(*************************************** EtherCAT Diag *********************************************)
(* generate Net Id *)
sEcMasterNetId := F_CreateAmsNetId(nIds := arrEcMasterNetId);
fbEtherCATDiag(
    sIPCNetID			:= '',
    sMasterNetID		:= sEcMasterNetId,
    nMasterDevID		:= nEcMasterDeviceId,
    nSlaveCount			:= nEcMasterSlaveCount,
    nSlaveCountCfg		:= nEcMasterSlaveCountCfg,
    nMasterDevState		:= nEcMasterDevState,
    bAllFrameWcStatesOK	:= bAllFrameWcStatesOK,
    tTimeout			:= T#5s,
    astDiagSlaveInfo	:= astDiagSlaveInfo,
    astDiagSlaveInfoScanned	:= astDiagSlaveInfoScanned,
    bEtherCATOK			=> bEtherCATOK,
    bFrameWcStateError	=> bFrameWcStateError,
    bSlaveCountError	=> bSlaveCountError,
    bMasterDevStateError=> bMasterDevStateError,
    stMasterDevState	=> stMasterDevState,
    bBusy				=> bBusy,
    bError				=> bError,
    nErrorID			=> nErrorID
);

END_FUNCTION_BLOCK

// ---- POUs/Diagnostics/FB_EtherCATFrameDiag.TcPOU
FUNCTION_BLOCK FB_EtherCATFrameDiag
VAR_INPUT
    nFrmXWcState 		: WORD;				// FrmXWcState
    nReqZeroMask 		: WORD := 16#FFFF;	// mask, bit TRUE: require wFrmXWcState.bit = FALSE, bit FALSE: ignore wFrmXWcState.bit *)
END_VAR
VAR_OUTPUT
    bFrameWcStateOK		: BOOL;				// result of fram state check
END_VAR
VAR
END_VAR

(* mask out ignored error bits and compare result against 0 *)
bFrameWcStateOK := ((nFrmXWcState AND nReqZeroMask) = 0);

END_FUNCTION_BLOCK

// ---- POUs/Diagnostics/FB_EtherCATDiag.TcPOU
FUNCTION_BLOCK FB_EtherCATDiag
VAR_INPUT
    sIPCNetID					: T_AmsNetId; 	// AmsNetId of the IPC
    sMasterNetID				: T_AmsNetId; 	// AmsNetId of the EtherCAT master device
    nMasterDevID				: UINT;			// Device ID of EtherCAT master
    nSlaveCount 				: UINT;			// current slave count
    nSlaveCountCfg 				: UINT;			// configured slave count
    nMasterDevState				: WORD;			// device state of EtherCAT Master
    bAllFrameWcStatesOK			: BOOL;			// all FrameWcState OK?
    tTimeout					: TIME := T#5S; // ads timeout
    eSubSystem : E_Subsystem := E_Subsystem.FIELDBUS; // Subsystem, change to (MPS, VACUUM, MOTION, etc)
END_VAR
VAR_OUTPUT
    bEtherCATOK					: BOOL;			// no problem on EtherCAT
    bFrameWcStateError			: BOOL;			// error in at least one frame
    bSlaveCountError			: BOOL;			// EtherCAT slave count mismatch (# of cfg slaves <> # of found slaves)
    bMasterDevStateError		: BOOL;			// error in master device state
    stMasterDevState			: ST_EcMasterDevState; // splitted master device state
    bBusy						: BOOL;			// FB busy
    bError						: BOOL;			// FB with error
    nErrorID					: UDINT;		// FB error ID
END_VAR
VAR_IN_OUT
    astDiagSlaveInfo 			: ARRAY [0..cnEscMaxPorts] OF ST_SlaveStateInfo;		// read in info from configured slaves
    astDiagSlaveInfoScanned		: ARRAY [0..cnEscMaxPorts] OF ST_SlaveStateInfoScanned;	// read in info from scanned slaves
END_VAR
VAR
    eState						: E_EcatDiagState;
    nMasterDevStatePrev			: WORD;
    bSlaveCountErrorPrev		: BOOL;
    bAllFrameWcStatesOKPrev		: BOOL;
    bDiagReq					: BOOL := TRUE;
    nI							: UDINT;
    nP							: UDINT;

    astSlaveInfo 				: ARRAY [0..cnSlaveAddrArrSize] OF ST_SlaveStateInfo;
    stSlaveInfo  :   REFERENCE TO ST_SlaveStateInfo;

    (* -- Get Slave Addresses *)
    fbGetSlaveAddresses 		: FB_EcGetAllSlaveAddr;
    anSlaveAddresses 			: ARRAY[0..cnSlaveAddrArrSize] OF UINT;
    nNumOfSlavesRead			: UINT;

    (* -- Get Slave States *)
    fbGetAllSlaveStates			: FB_EcGetAllSlaveStates;
    astSlaveStates 				: ARRAY[0..cnSlaveAddrArrSize] OF ST_EcSlaveState;

    (* -- Get Topology Data *)
    nTopologyData				: UDINT;
    fbGetTopologyData			: ADSREAD;
    astTopologyData				: ARRAY[0..cnSlaveAddrArrSize] OF ST_TopologyData;

    (* -- Check Topology *)
    anDiagIndex					: ARRAY [0..cnEscMaxPorts] OF UINT;
    nDiagIndex : UINT;
    anDiagPort					: ARRAY [0..cnEscMaxPorts] OF UINT;
    nDiagPort : UINT;
    nIdx						: DINT;

    (* -- Scan Slaves *)
    fbEcGetScannedSlaves		: FB_EcGetScannedSlaves;
    astScannedSlaveInfo			: ARRAY [0..cnSlaveAddrArrSize] OF ST_EcSlaveScannedData; // what...
    rScannedSlaveInfo   :   REFERENCE TO ST_EcSlaveScannedData;
    nScannedSlaves				: UINT;

    (* -- Get Slave Identities *)
    fbGetSlaveIdentity			: FB_EcGetSlaveIdentity;
    stIdentity 					: ST_EcSlaveIdentity;

    (* -- Get Slave Names *)
    fbGetSlaveName 				: IOF_GetBoxNameByAddr;
    astSlaveInfoScanned			: ARRAY [0..cnSlaveAddrArrSize] OF ST_SlaveStateInfoScanned; // the F
    stSlaveInfoScanned   :   REFERENCE TO ST_SlaveStateInfoScanned;
    sStringName						: STRING;



    // Logging components
    fbLogger : FB_LogMessage := (eSubsystem := eSubsystem);

    fbJson : FB_JsonSaxWriter;
    fbJsonDataType : FB_JsonReadWriteDataType;
    stDiagSlaveInfo : REFERENCE TO ST_SlaveStateInfo;
    fbEtherCATOK : F_TRIG;
    fbFrameWcStateError : R_TRIG;
    fbMasterError : R_TRIG;
    nJsonIdx : UINT;
    {attribute 'analysis' := '-27'}
    sTest : T_MaxString;
END_VAR

(* cyclic diag *)
bFrameWcStateError := NOT bAllFrameWcStatesOK;

bSlaveCountError := (nSlaveCount <> nSlaveCountCfg) OR (nSlaveCount = 0);
IF (bSlaveCountError AND NOT bSlaveCountErrorPrev) OR (NOT bSlaveCountError AND bSlaveCountErrorPrev) THEN
    bSlaveCountErrorPrev := bSlaveCountError;
    bDiagReq := TRUE; // slave count error change detected --> diag required
END_IF

IF (bAllFrameWcStatesOK AND NOT bAllFrameWcStatesOKPrev) OR (NOT bAllFrameWcStatesOK AND bAllFrameWcStatesOKPrev) THEN
    bAllFrameWcStatesOKPrev := bAllFrameWcStatesOK;
    bDiagReq := TRUE; // frame error change detected --> diag required
END_IF

IF (nMasterDevState <> nMasterDevStatePrev) THEN
    M_CheckMasterDevState();
    bDiagReq := TRUE; // devstate change detected --> diag required
END_IF

(* acyclic diag *)
CASE eState OF
E_EcatDiagState.Idle: (* IDLE *)
    IF bDiagReq THEN				// diag requested
        bDiagReq := FALSE;

        IF sMasterNetID <> '' AND sMasterNetID <> '0.0.0.0.0.0' THEN
            eState := E_EcatDiagState.GetSlaveAddresses;	// execute diag
            bBusy := TRUE;
        ELSE
            bError := TRUE;
            nErrorID := 7;
        END_IF

        bEtherCATOK := FALSE;
    ELSE
        // check for changes in idle
        IF (bSlaveCountError OR bMasterDevStateError OR NOT bAllFrameWcStatesOK) AND NOT (astSlaveInfo[anDiagIndex[0]].bDiagData) THEN
            bEtherCATOK := FALSE;
            bDiagReq := TRUE;//new error --> diag requested
        ELSIF (bSlaveCountError AND NOT bSlaveCountErrorPrev) OR (NOT bSlaveCountError AND bSlaveCountErrorPrev) THEN
            bSlaveCountErrorPrev := bSlaveCountError;
            bEtherCATOK := FALSE;
            bDiagReq := TRUE;// slave count error change detected --> diag required
        ELSIF (nMasterDevState <> nMasterDevStatePrev) THEN
            bEtherCATOK := FALSE;
            bDiagReq := TRUE;// devstate change detected --> diag required
        ELSIF (bAllFrameWcStatesOK AND NOT bAllFrameWcStatesOKPrev) OR (NOT bAllFrameWcStatesOK AND bAllFrameWcStatesOKPrev) THEN
            bAllFrameWcStatesOKPrev := bAllFrameWcStatesOK;
            bEtherCATOK := FALSE;
            bDiagReq := TRUE;// frame error change detected --> diag required
        ELSIF (bSlaveCountError OR bMasterDevStateError OR NOT bAllFrameWcStatesOK OR astSlaveInfo[anDiagIndex[0]].bDiagData) THEN
            bEtherCATOK := FALSE;
        ELSE
            bEtherCATOK := TRUE;
        END_IF
    END_IF

E_EcatDiagState.GetSlaveAddresses: (* get adresses *)
    M_GetSlaveAdresses();

E_EcatDiagState.GetSlaveStates: (* get states *)
    M_GetSlaveStates();

E_EcatDiagState.GetTopoDataLen:	(* get topology data length *)
    M_GetTopoDataLen();

E_EcatDiagState.GetTopoData:	(* get topology data *)
    M_GetTopoData();

E_EcatDiagState.ScanSlaves:	(* scan slaves *)
    M_ScanSlaves();

E_EcatDiagState.GetSlaveIdentity:	(* get identity *)
    M_GetSlaveIdentity();

E_EcatDiagState.GetSlaveName:	(* get name *)
    M_GetSlaveName();

E_EcatDiagState.GetScannedSlaveName:	(* get scanned name *)
    M_GetScannedSlaveName();

E_EcatDiagState.LogDiagnostics: (* Log diagnostics *)
    (* I can't get the fbJsonDataType to actually convert the slave info
    structures. I just get nulls. Either I am doing this wrong, or when
    the symbol parser encounters datatypes it can't deal with it nulls
    the whole thing. I'll keep this code commented out until someone figures
    out how to deal with parsing the slave structs into the json payload *)
    IF nJsonIdx < nNumOfSlavesRead THEN // the last entry is always blank
        nJsonIdx := MIN(cnSlaveAddrArrSize, nJsonIdx);
        stDiagSlaveInfo REF= astSlaveInfo[nJsonIdx];
        DiagnosticJson();
        fbLogger(sMsg:=CONCAT('Diag Results: ', stDiagSlaveInfo.sName),
                eSevr:=TcEventSeverity.Info);
        nJsonIdx := nJsonIdx + 1;
    ELSE
        nJsonIdx := 0;
        eState := E_EcatDiagState.Done;
    END_IF

E_EcatDiagState.Done:	(* DONE *)
    bBusy := FALSE;
    eState := 0;

END_CASE

// Log messages
fbEtherCATOK(CLK:=bEtherCATOK);
IF fbEtherCATOK.Q THEN
    fbLogger(sMsg:='EtherCAT failure, starting diagnostic', eSevr:=TcEventSeverity.Critical, sJson:='');
END_IF

fbFrameWcStateError(CLK:=bFrameWcStateError);
IF fbFrameWcStateError.Q THEN
    fbLogger(sMsg:='Working Counter Frame Error: error in at least one frame', eSevr:=TcEventSeverity.Error, sJson:='');
END_IF

fbMasterError(CLK:=bMasterDevStateError);
IF fbMasterError.Q THEN
    fbJson.StartObject();
        fbJson.AddKey('ecat_master_diag');
        fbJson.StartObject();
            fbJson.AddKey('bAtLeastOneNotInOp');
            fbJson.AddBool(stMasterDevState.bAtLeastOneNotInOp);
            fbJson.AddKey('bDcNotInSync');
            fbJson.AddBool(stMasterDevState.bDcNotInSync);
            fbJson.AddKey('bDriverNotFound');
            fbJson.AddBool(stMasterDevState.bDriverNotFound);
            fbJson.AddKey('bLinkError');
            fbJson.AddBool(stMasterDevState.bLinkError);
            fbJson.AddKey('bMissFrmRedMode');
            fbJson.AddBool(stMasterDevState.bMissFrmRedMode);
            fbJson.AddKey('bResetActive');
            fbJson.AddBool(stMasterDevState.bResetActive);
            fbJson.AddKey('bResetRequired');
            fbJson.AddBool(stMasterDevState.bResetRequired);
            fbJson.AddKey('bWatchdogTriggerd');
            fbJson.AddBool(stMasterDevState.bWatchdogTriggerd);
            fbJson.AddKey('eEcState');
            fbJson.AddUdint(stMasterDevState.eEcState);
        fbJson.EndObject();
    fbJson.EndObject();
    fbJson.CopyDocument(fbLogger.sJson, SIZEOF(fbLogger.sJson));
    fbLogger(sMsg:='Master error: error in master device state', eSevr:=TcEventSeverity.Critical);
    fbJson.ResetDocument();
END_IF

ACTION DiagnosticJson:
fbJson.StartObject();
    fbJson.AddKey('ecat_diag');
    fbJson.StartObject();

        fbJson.AddKey('nECAddr');
        fbJson.AddUdint(stDiagSlaveInfo.nECAddr);

        fbJson.AddKey('nIndex');
        fbJson.AddDint(stDiagSlaveInfo.nIndex);

        fbJson.AddKey('sName');
        fbJson.AddString(stDiagSlaveInfo.sName);

        fbJson.AddKey('sType');
        fbJson.AddString(stDiagSlaveInfo.sType);

        fbJson.AddKey('bDiagData');
        fbJson.AddBool(stDiagSlaveInfo.bDiagData);

        fbJson.AddKey('stPortCRCErrors');
        fbjson.StartObject();

            fbJson.AddKey('portA');
            fbJson.AddUdint(stDiagSlaveInfo.stPortCRCErrors.portA);
            fbJson.AddKey('portB');
            fbJson.AddUdint(stDiagSlaveInfo.stPortCRCErrors.portB);
            fbJson.AddKey('portC');
            fbJson.AddUdint(stDiagSlaveInfo.stPortCRCErrors.portC);
            fbJson.AddKey('portD');
            fbJson.AddUdint(stDiagSlaveInfo.stPortCRCErrors.portD);

        fbJson.EndObject();

        fbJson.AddKey('nSumCRCErrors');
        fbjson.AddUdint(stDiagSlaveInfo.nSumCRCErrors);

        fbJson.AddKey('stState');
        fbJson.StartObject();

            fbJson.AddKey('eEcState ');
            fbJson.AddUdint(stDiagSlaveInfo.stState.eEcState);
            fbJson.AddKey('nReserved');
            fbJson.AddUdint(stDiagSlaveInfo.stState.nReserved);
            fbJson.AddKey('bError');
            fbJson.AddBool(stDiagSlaveInfo.stState.bError);
            fbJson.AddKey('bInvalidVPRS');
            fbJson.AddBool(stDiagSlaveInfo.stState.bInvalidVPRS);
            fbJson.AddKey('nReserved2');
            fbJson.AddUdint(stDiagSlaveInfo.stState.nReserved2);
            fbJson.AddKey('bNoCommToSlave');
            fbJson.AddBool(stDiagSlaveInfo.stState.bNoCommToSlave);
            fbJson.AddKey('bLinkError');
            fbJson.AddBool(stDiagSlaveInfo.stState.bLinkError);
            fbJson.AddKey('bMissingLink');
            fbJson.AddBool(stDiagSlaveInfo.stState.bMissingLink);
            fbJson.AddKey('bUnexpectedLink');
            fbJson.AddBool(stDiagSlaveInfo.stState.bUnexpectedLink);
            fbJson.AddKey('bPortA');
            fbJson.AddBool(stDiagSlaveInfo.stState.bPortA);
            fbJson.AddKey('bPortB');
            fbJson.AddBool(stDiagSlaveInfo.stState.bPortB);
            fbJson.AddKey('bPortC');
            fbJson.AddBool(stDiagSlaveInfo.stState.bPortC);
            fbJson.AddKey('bPortD');
            fbJson.AddBool(stDiagSlaveInfo.stState.bPortD);

        fbJson.EndObject();

    fbJson.EndObject();

fbJson.EndObject();

fbJson.CopyDocument(fbLogger.sJson, SIZEOF(fbLogger.sJson));
fbJson.ResetDocument();
END_ACTION

ACTION M_CheckMasterDevState:
(* check master errors based on devstate *)
bMasterDevStateError 				:= nMasterDevState <> 0;
stMasterDevState.bLinkError 		:= ((nMasterDevState AND 16#000F) = 1) OR ((nMasterDevState AND 16#000F) = 4);
stMasterDevState.bResetRequired 	:= ((nMasterDevState AND 16#000F) = 2) OR ((nMasterDevState AND 16#FFF0) = 16#10);
stMasterDevState.bMissFrmRedMode 	:= (nMasterDevState AND 16#000F) = 8;
stMasterDevState.bWatchdogTriggerd 	:= (nMasterDevState AND 16#20) = 16#20;
stMasterDevState.bDriverNotFound 	:= (nMasterDevState AND 16#40) = 16#40;
stMasterDevState.bResetActive 		:= (nMasterDevState AND 16#80) = 16#80;
stMasterDevState.bAtLeastOneNotInOp := ((nMasterDevState AND 16#100) = 16#100) OR ((nMasterDevState AND 16#200) = 16#200) OR
                                        ((nMasterDevState AND 16#400) = 16#400) OR ((nMasterDevState AND 16#800) = 16#800);
stMasterDevState.bDcNotInSync 		:= (nMasterDevState AND 16#1000) = 16#1000;
nMasterDevStatePrev 				:= nMasterDevState;
END_ACTION

ACTION M_GetScannedSlaveName:

stSlaveInfoScanned REF= astSlaveInfoScanned[anDiagIndex[nIdx]];
rScannedSlaveInfo REF= astScannedSlaveInfo[anDiagIndex[nIdx]];

fbGetSlaveName(
    NETID		:= sIPCNetId,
    DEVICEID	:= nMasterDevID,
    BOXADDR		:= rScannedSlaveInfo.nAddr,
    START		:= TRUE,
    TMOUT		:= tTimeout,
    BOXNAME		=> sStringName
);

IF NOT fbGetSlaveName.BUSY THEN
    fbGetSlaveName(START:= FALSE);

    (* add scanned info *)
    stSlaveInfoScanned.nIndex 	:= nDiagIndex + 1;
    IF rScannedSlaveInfo.nAddr <> 0 THEN
        IF NOT fbGetSlaveName.ERR THEN
            stSlaveInfoScanned.sName := sStringName;
        END_IF
    ELSE
        stSlaveInfoScanned.sType		:= '';
    END_IF

    IF (nDiagIndex < nScannedSlaves) THEN
        stSlaveInfoScanned.sType		:= F_ConvProductCodeToString(rScannedSlaveInfo.stSlaveIdentity);
    ELSE
        stSlaveInfoScanned.sType		:= '';
    END_IF

    stSlaveInfoScanned.nECAddr	:= rScannedSlaveInfo.nAddr;

    IF stSlaveInfoScanned.sName <> stSlaveInfo.sName THEN
        stSlaveInfoScanned.bDifferentName := TRUE;
    ELSE
        stSlaveInfoScanned.bDifferentName := FALSE;
    END_IF

    IF stSlaveInfoScanned.nECAddr <> stSlaveInfo.nECAddr THEN
        stSlaveInfoScanned.bDifferentAddr := TRUE;
    ELSE
        stSlaveInfoScanned.bDifferentAddr := FALSE;
    END_IF

    IF stSlaveInfoScanned.sType <> stSlaveInfo.sType THEN
        stSlaveInfoScanned.bDifferentType := TRUE;
    ELSE
        stSlaveInfoScanned.bDifferentType := FALSE;
    END_IF

    IF nIdx < cnEscMaxPorts THEN
        nIdx := nIdx + 1;
        eState := E_EcatDiagState.GetSlaveIdentity; // loop back
    ELSE
        nIdx := 0;
        eState := E_EcatDiagState.LogDiagnostics;

        FOR nI := 0 TO cnEscMaxPorts DO
            IF anDiagPort[nI] <> 0 THEN
                astDiagSlaveInfo[nI] := astSlaveInfo[anDiagIndex[nI]];
                astDiagSlaveInfoScanned[nI] := astSlaveInfoScanned[anDiagIndex[nI]];
            ELSE
                MEMSET(ADR(astDiagSlaveInfo[nI]), 0, SIZEOF(astDiagSlaveInfo[nI]));
                MEMSET(ADR(astDiagSlaveInfoScanned[nI]), 0, SIZEOF(astDiagSlaveInfoScanned[nI]));
            END_IF
        END_FOR
    END_IF
END_IF
END_ACTION

ACTION M_GetSlaveAdresses:
fbGetSlaveAddresses(
    sNetId		:= sMasterNetID,
    pAddrBuf	:= ADR(anSlaveAddresses),
    cbBufLen	:= SIZEOF(anSlaveAddresses),
    bExecute	:= TRUE,
    tTimeout	:= tTimeout,
    nSlaves		=> nNumOfSlavesRead
);

IF NOT fbGetSlaveAddresses.bBusy THEN
    fbGetSlaveAddresses(bExecute:= FALSE);
    IF NOT fbGetSlaveAddresses.bError THEN
        FOR nI := 0 TO MIN(nNumOfSlavesRead, cnSlaveAddrArrSize) DO
            astSlaveInfo[nI].nECAddr := anSlaveAddresses[nI];
        END_FOR
    END_IF
    eState := GetSlaveStates;
END_IF
END_ACTION

ACTION M_GetSlaveIdentity:

nDiagIndex := anDiagIndex[nIdx];
nDiagPort := anDiagPort[nIdx];

stSlaveInfo REF= astSlaveInfo[nDiagIndex];

fbGetSlaveIdentity(
    sNetId		:= sMasterNetID,
    nSlaveAddr	:= stSlaveInfo.nECAddr,
    bExecute	:= TRUE,
    tTimeout	:= tTimeout,
    identity	=> stIdentity
);

IF NOT fbGetSlaveIdentity.bBusy THEN
    fbGetSlaveIdentity(bExecute:= FALSE);

    IF NOT fbGetSlaveIdentity.bError THEN
        IF anDiagPort[nIdx] <> 0 THEN
            stSlaveInfo.nIndex	:= anDiagIndex[nIdx] + 1;
            stSlaveInfo.sType 	:= F_ConvProductCodeToString(stSlaveIdentity := stIdentity);
        END_IF
    END_IF
    eState := E_EcatDiagState.GetSlaveName;
END_IF
END_ACTION

ACTION M_GetSlaveName:
fbGetSlaveName(
    NETID		:= sIPCNetId,
    DEVICEID	:= nMasterDevID,
    BOXADDR		:= stSlaveInfo.nECAddr,
    START		:= TRUE,
    TMOUT		:= tTimeout,
    BOXNAME		=> sStringName
);

IF NOT fbGetSlaveName.BUSY THEN
    fbGetSlaveName(START:= FALSE);

    IF NOT fbGetSlaveName.ERR THEN
        IF nDiagPort <> 0 THEN
            stSlaveInfo.sName 	:= sStringName;
        END_IF
    END_IF

    eState := E_EcatDiagState.GetScannedSlaveName;
END_IF
END_ACTION

ACTION M_GetSlaveStates:
fbGetAllSlaveStates(
    sNetId		:= sMasterNetID,
    pStateBuf	:= ADR(astSlaveStates),
    cbBufLen	:= SIZEOF(astSlaveStates),
    bExecute	:= TRUE,
    tTimeout	:= tTimeout,
    nSlaves		=> nNumOfSlavesRead
);

IF NOT fbGetAllSlaveStates.bBusy THEN
    fbGetAllSlaveStates(bExecute:= FALSE);

    IF NOT fbGetAllSlaveStates.bError THEN
        IF nNumOfSlavesRead = nSlaveCountCfg THEN
            FOR nI := 0 TO cnEscMaxPorts DO
                anDiagIndex[nI] := 0;
            END_FOR

            (* split slave state and link state *)
            FOR nI := 0 TO MIN(nNumOfSlavesRead, cnSlaveAddrArrSize) DO
                (* slave state*)
                astSlaveInfo[nI].stState.eEcState 		:= astSlaveStates[nI].deviceState AND 16#0F;
                astSlaveInfo[nI].stState.bError 			:= astSlaveStates[nI].deviceState.4;
                astSlaveInfo[nI].stState.bInvalidVPRS 	:= astSlaveStates[nI].deviceState.5;
                (* link state *)
                astSlaveInfo[nI].stState.bNoCommToSlave 	:= astSlaveStates[nI].linkState.0;
                astSlaveInfo[nI].stState.bLinkError 		:= astSlaveStates[nI].linkState.1;
                astSlaveInfo[nI].stState.bMissingLink 	:= astSlaveStates[nI].linkState.2;
                astSlaveInfo[nI].stState.bUnexpectedLink := astSlaveStates[nI].linkState.3;
                astSlaveInfo[nI].stState.bPortA 			:= astSlaveStates[nI].linkState.4;
                astSlaveInfo[nI].stState.bPortB 			:= astSlaveStates[nI].linkState.5;
                astSlaveInfo[nI].stState.bPortC 			:= astSlaveStates[nI].linkState.6;
                astSlaveInfo[nI].stState.bPortD 			:= astSlaveStates[nI].linkState.7;
                (* DiagData *)
                astSlaveInfo[nI].bDiagData	:= ((astSlaveStates[nI].deviceState AND 16#F0) <> 0) OR
                    (((astSlaveStates[nI].deviceState AND 16#0F) > 0) AND ((astSlaveStates[nI].deviceState AND 16#0F) < 8)) OR
                    (astSlaveStates[nI].linkState <> 0);

                IF astSlaveInfo[nI].bDiagData THEN
                    IF (nI=0) THEN
                        anDiagIndex[0] := 0;
                    ELSE
                        IF (anDiagIndex[0] = 0) AND NOT astSlaveInfo[0].bDiagData THEN
                            anDiagIndex[0] :=  UDINT_TO_UINT(nI);
                        END_IF
                    END_IF
                END_IF
            END_FOR
        END_IF
    END_IF

    IF astSlaveInfo[anDiagIndex[0]].bDiagData THEN
        eState := E_EcatDiagState.GetTopoDataLen;
    ELSE
        FOR nI := 0 TO cnEscMaxPorts DO
            MEMSET(ADR(astDiagSlaveInfo[nI]), 0, SIZEOF(astDiagSlaveInfo[nI]));
            MEMSET(ADR(astDiagSlaveInfoScanned[nI]), 0, SIZEOF(astDiagSlaveInfoScanned[nI]));
        END_FOR
        eState := E_EcatDiagState.Done;
    END_IF
END_IF
END_ACTION

ACTION M_GetTopoData:
fbGetTopologyData(
    NETID	:= sMasterNetID,
    PORT	:= 16#FFFF,
    IDXGRP	:= 16#22,
    IDXOFFS	:= 0,
    LEN		:= nTopologyData*SIZEOF(astTopologyData[0]),
    DESTADDR:= ADR(astTopologyData),
    READ	:= TRUE,
    TMOUT	:= tTimeout,
);

IF NOT fbGetTopologyData.BUSY THEN
    fbGetTopologyData(READ := FALSE);

    IF NOT fbGetTopologyData.ERR THEN
        anDiagPort[0] := astTopologyData[anDiagIndex[0]].nOwnPhysicalAddr;
        anDiagPort[1] := astTopologyData[anDiagIndex[0]].stPhysicalAddr.portB;
        anDiagPort[2] := astTopologyData[anDiagIndex[0]].stPhysicalAddr.portC;
        anDiagPort[cnEscMaxPorts] := astTopologyData[anDiagIndex[0]].stPhysicalAddr.portD;

        (* clear diag index  *)
        anDiagIndex[1] := 0;
        anDiagIndex[2] := 0;
        anDiagIndex[cnEscMaxPorts] := 0;

        (* find slaves on PortB-D of first slave with diag *)
        FOR nP := 0 TO cnEscMaxPorts DO
            IF anDiagPort[nP] <> 0 THEN
            FOR nI := 0 TO MIN(nTopologyData-1,cnSlaveAddrArrSize) DO
                IF astTopologyData[nI].nOwnPhysicalAddr = anDiagPort[nP] THEN
                    anDiagIndex[nP] := UDINT_TO_UINT(nI);
                    EXIT;
                END_IF
            END_FOR
        END_IF
        END_FOR
    END_IF

    nIdx := 0;
    eState := E_EcatDiagState.ScanSlaves;
END_IF
END_ACTION

ACTION M_GetTopoDataLen:
fbGetTopologyData(
    NETID	:= sMasterNetID,
    PORT	:= 16#FFFF,
    IDXGRP	:= EC_ADS_IGRP_MASTER_COUNT_SLAVE,
    IDXOFFS	:= EC_ADS_IOFFS_MASTER_COUNT_SLAVE,
    LEN		:= SIZEOF(nTopologyData),
    DESTADDR:= ADR(nTopologyData),
    READ	:= TRUE,
    TMOUT	:= tTimeout,
);

IF NOT fbGetTopologyData.BUSY THEN
    fbGetTopologyData(READ := FALSE);

    eState := E_EcatDiagState.GetTopoData;
END_IF
END_ACTION

ACTION M_ScanSlaves:
fbEcGetScannedSlaves(
    bExecute				:= TRUE,
    sNetId					:= sMasterNetID,
    pArrEcScannedSlaveInfo	:= ADR(astScannedSlaveInfo),
    cbBufLen				:= SIZEOF(astScannedSlaveInfo),
    tTimeout				:= tTimeout
);

IF NOT fbEcGetScannedSlaves.bBusy THEN
    fbEcGetScannedSlaves(bExecute := FALSE);

    IF fbEcGetScannedSlaves.bError THEN
        nScannedSlaves := 0;
    ELSE
        nScannedSlaves := fbEcGetScannedSlaves.nSlaves;
    END_IF

    eState := E_EcatDiagState.GetSlaveIdentity;

END_IF
END_ACTION

END_FUNCTION_BLOCK

// ---- POUs/EPS/FB_EPS.TcPOU
FUNCTION_BLOCK FB_EPS
VAR_IN_OUT
    eps : DUT_EPS;
END_VAR
VAR_OUTPUT
END_VAR
VAR
END_VAR

METHOD setBit : BOOL
VAR_INPUT
    nBits : BYTE;
    bValue : BOOL;
END_VAR
VAR
    nMask : UDINT := 1;
    nBitValue : UDINT := 0;
END_VAR
nMask := SHL(nMask, nBits);
// Checking the VAR_IN_OUT reference, leave the current method in case of invalid reference
IF NOT __ISVALIDREF(eps) THEN
    RETURN;
END_IF

(* Access to VAR_IN_OUT reference (only if the reference was confirmed as valid before) *)
nBitValue := SHR((nMask AND eps.nFlags), nBits);

IF (TO_BOOL(nBitValue)) <> bValue THEN
    eps.nFlags := eps.nFlags XOR nMask;
END_IF

// Check if all values are true
IF eps.nFlags = 16#FFFFFFFF THEN
    eps.bEPS_OK := TRUE;
ELSE
    eps.bEPS_OK := FALSE;
END_IF
END_METHOD

METHOD setDescription : BOOL
VAR_INPUT
    desciption : STRING;
END_VAR

// Checking the VAR_IN_OUT reference, leave the current method in case of invalid reference
IF NOT __ISVALIDREF(eps) THEN
    RETURN;
END_IF

(* Access to VAR_IN_OUT reference (only if the reference was confirmed as valid before) *)
eps.sFlagDesc := desciption;
END_METHOD

METHOD setMessage : BOOL
VAR_INPUT
    message : STRING;
END_VAR
// Checking the VAR_IN_OUT reference, leave the current method in case of invalid reference
IF NOT __ISVALIDREF(eps) THEN
    RETURN;
END_IF
// Access to VAR_IN_OUT reference (only if the reference was confirmed as valid before)
eps.sMessage := message;
END_METHOD

END_FUNCTION_BLOCK

// ---- POUs/Functions/FB_EcatDiag.TcPOU
(*
Ecat bus diagnostic tool
2015-11-4 Alex Wallace
This function block checks the states of all slaves on the ecat bus network,
it could be modified to export the states of the slaves on an individual basis,
but for now it sets the output boolean true if all slaves are OP and false otherwise.
To start the block provide a falling edge on the first pass boolean input.

2018-05-05 Margaret Ghaly
Function block has been modified to retrieve the Device State of the Ethercat Master.
It also exports the states and information of each individual configured Slave.
And saves them in the array q_aEcConfSlaveInfo.
*)
FUNCTION_BLOCK FB_EcatDiag
VAR_INPUT
    {attribute 'naming' := 'omit'}
    I_AMSNetId AT %I* : AMSNETID; //Link to the AMSNETID name in the ethercat master info.
    bFirstPass: BOOL; //Hook to system first pass boolean for proper initialization (must be true for the first cycle of the PLC)
END_VAR
VAR_OUTPUT
    bAllSlaveStatesGood: BOOL; // Set to True if all Slaves are in OP State
    anTermStates: ARRAY[1..256] OF BYTE; //ECAT State of terminals in the bus
    bMasterStateGood:BOOL; // Set to True if the Master Device State is OP
    nMasterState: WORD; // The Device State of the Master
    sMasterState:STRING; //State of the ECAT master
    astEcConfSlaveInfo :  ARRAY[1..256] OF ST_EcDevice; //State of all ECAT slaves in the bus
    nSlaves: UINT; // the Number of the connected Slaves
END_VAR
VAR
    sNetId: T_AmsNetId; //NetId string
    astTermStates: ARRAY[1..256] OF ST_EcSlaveState; //ECAT Slave States Buffer
    astEcConfSlaveInfoLocal: ARRAY[1..256] OF ST_EcSlaveConfigData; //ECAT Slave Configs Buffer
    fbGetAllSlaveStates: FB_EcGetAllSlaveStates; //Acquires the ECAT Slave States puts them into astTermStates

    fbGetMasterState: FB_EcGetMasterState; //Acquires ECAT Master State
    fbGetConfSlaves: FB_EcGetConfSlaves; //Acquires the ECAT slave configuration of the bus (how many, what kind, etc)
    {attribute 'naming' := 'omit'}
    ftReset: F_TRIG; //Reset trigger sensor
    {attribute 'naming' := 'omit'}
    ftMasterReset: F_TRIG; //Retrigger sensor for GetMasterState
    nIterator: INT; //Generic iterator placeholder
END_VAR

//Create the net ID string
sNetId := F_CreateAmsNetId(I_AMSNetId);

//Query the state of all terminals, collect in astTermStates
ftReset(CLK:=fbGetAllSlaveStates.bBusy OR bFirstPass);
fbGetAllSlaveStates.bExecute := ftReset.Q;
fbGetAllSlaveStates(sNetId:=sNetId, pStateBuf := ADR(astTermStates), cbBufLen:=SIZEOF(astTermStates));
//Keep checking...



//Cycle through each entry in the array and check if we have anyone not in OP and that the link state is good.
// If so, then set our global IO bad boolean.
IF fbGetAllSlaveStates.nSlaves > 0 THEN
    bAllSlaveStatesGood := TRUE;
FOR nIterator := 1 TO (UINT_TO_INT(fbGetAllSlaveStates.nSlaves) ) BY 1
    DO
    IF NOT( (astTermStates[nIterator].deviceState = EC_DEVICE_STATE_OP) AND (astTermStates[nIterator].linkState = EC_LINK_STATE_OK)) THEN
        bAllSlaveStatesGood := FALSE;
    END_IF
    anTermStates[nIterator] := astTermStates[nIterator].deviceState;
    astEcConfSlaveInfo[nIterator].nDeviceState :=astTermStates[nIterator].deviceState;//
    astEcConfSlaveInfo[nIterator].nLinkState :=astTermStates[nIterator].linkState;//
    astEcConfSlaveInfo[nIterator].sDeviceState:= F_ConvSlaveStateToString(state:=astTermStates[nIterator]);//

END_FOR
END_IF

// Read the EtherCAT state of the master. If the call is successful,
//the State output variable of type WORD contains the requested status information.
ftMasterReset(CLK:=fbGetMasterState.bBusy OR bFirstPass);
fbGetMasterState(sNetId:= sNetId, bExecute:=ftMasterReset.Q,
                state => nMasterState,bError=>,
                nErrId=>);
bMasterStateGood:= (fbGetMasterState.state = BYTE_TO_UINT(EC_DEVICE_STATE_OP));
sMasterState := F_ConvMasterDevStateToString(fbGetMasterState.state);

//This function is used to read a list of all configured slaves from the EtherCat master object Directory
//needs to run only once
fbGetConfSlaves(bExecute := bFirstPass, sNetId :=sNetId, pArrEcConfSlaveInfo := ADR(astEcConfSlaveInfoLocal),cbBufLen := SIZEOF(astEcConfSlaveInfoLocal));
nSlaves:=fbGetConfSlaves.nSlaves;

IF  NOT (fbGetConfSlaves.bBusy) THEN
    FOR nIterator := 1 TO (UINT_TO_INT(fbGetConfSlaves.nSlaves) ) BY 1
    DO
    astEcConfSlaveInfo[nIterator].nAddrr :=astEcConfSlaveInfoLocal[nIterator].nAddr;
    astEcConfSlaveInfo[nIterator].sName :=astEcConfSlaveInfoLocal[nIterator].sName;
    astEcConfSlaveInfo[nIterator].sType :=astEcConfSlaveInfoLocal[nIterator].sType;
END_FOR
    fbGetConfSlaves.bExecute := FALSE;
END_IF

END_FUNCTION_BLOCK

// ---- POUs/Functions/FB_Index.TcPOU
(* Index FB
A. Wallace 2016-9-3

Why doesn't beckhoff have this as a builtin type?

Use this thing to have a simple indexer with rollover.

*)
FUNCTION_BLOCK FB_Index
VAR_INPUT
    {attribute 'naming' := 'off'}
    LowerLimit : INT := 1; //Incrementer will rollver over to this value (and initialize to this value)
    ValInc : INT := 1; //Incrementer increments by this value
    UpperLimit	:	INT := 1; //Incrementer will rollover at this value to lower limit
    {attribute 'naming' := 'off'}
END_VAR
VAR_OUTPUT

END_VAR
VAR
    nVal	:	INT := LowerLimit; //Internal incrementer value, initialized to LowerLimit
END_VAR

{analysis -2} //Only the methods and actions are needed

ACTION Dec:
nVal := nVal - ValInc;
IF nVal < LowerLimit THEN nVal := UpperLimit; END_IF
END_ACTION

//Decrement the counter and return new value
METHOD DecVal : INT
VAR_INPUT
END_VAR
Dec();
DecVal := nVal;
END_METHOD

ACTION Inc:
// Dont use this, use ValInc
nVal := nVal + ValInc;
IF nVal >  UpperLimit THEN nVal := LowerLimit; END_IF
END_ACTION

//Increment the counter and return new value
METHOD PUBLIC IncVal : INT
VAR_INPUT
END_VAR
Inc();
IncVal := nVal;
END_METHOD

END_FUNCTION_BLOCK

// ---- POUs/Functions/FB_UnixTimeStampGlobal.TcPOU
FUNCTION_BLOCK FB_UnixTimeStampGlobal
(*
    Runs FB_UnixTimeStamp and stuffs the result into this library's GVL
    2019-10-09 Zachary Lentz
*)
VAR_INPUT
    // If TRUE, we will update the output on this cycle.
    bExecute: BOOL;
END_VAR
VAR_OUTPUT
END_VAR
VAR
    fbTimeStamp: FB_UnixTimeStamp;
END_VAR

fbTimeStamp(
    bExecute := bExecute,
    fTime => DefaultGlobals.fTimeStamp);

END_FUNCTION_BLOCK

// ---- POUs/Functions/FB_XKoyoPLCModbus.TcPOU
//Facilitates communication between Beckhoff and Koyo PLC over the network.
FUNCTION_BLOCK FB_XKoyoPLCModbus
VAR
    fbKoyo_PLCInputCoilsRx	:	FB_MBReadCoils; //FB for reading the coils from the other PLC
    anKoyo_PLC_CnBits	:	ARRAY [0..20] OF BYTE; //Buffer for coil readbacks
    {attribute 'naming' := 'omit'}
    ftReset	: F_TRIG; //Reset edge sensor
    {attribute 'naming' := 'omit'}
    tonRetry : TON; //Retry timer
    nIndex : INT; //Index for clearing the coil array
END_VAR
VAR_INPUT
    tRetryTime : TIME := T#10S; //Retry time if modbus transaction fails
    sIPAddr	 : STRING[15]; //IP address of the Koyo PLC
END_VAR
VAR_OUTPUT
    bNoPLCResponse : BOOL := TRUE; //Could not reach the PLC if true
    anPLCResponse   : ARRAY [0..20] OF BYTE; //Buffer of coils retrieved from the other PLC
    bError         : BOOL := FALSE; //Transaction or other error
END_VAR

(* Look ma' no wires! *)
(* A. Wallace, 2015-7-22
XKoyoPLCModbus

Facilitates communication between Beckhoff and Koyo PLC over the network.

Useful if you don't have time to run a wire. Fairly reliable.

*)

(* Modbus Info for Koyo
Modbus Addresses for
Koyo DL05/06/240/250/260/430/440/450 PLCs
PLC Memory Type		| Modbus start address Decimal (octal) | Function codes
Inputs (X)			  2048 (04000)							2
Special Relays (SP)	  3072 (06000)							2
Outputs (Y)			  2048 (04000)							1, 5, 15
Control Relays (C)	  3072 (06000)							1, 5, 15
Timer Contacts (T)	  6144 (014000)							1, 5, 15
Counter Contacts (CT) 6400 (014400)							1, 5, 15
Stage Status Bits (S) 6144 (012000)							1, 5, 15
*)

(* Begin code *)
// Retry after some time
tonRetry.IN := NOT fbKoyo_PLCInputCoilsRx.bBusy;
tonRetry.PT := tRetryTime;
tonRetry();

ftReset(CLK:=fbKoyo_PLCInputCoilsRx.bBusy);
ftReset();

fbKoyo_PLCInputCoilsRx.bExecute := ftReset.Q OR tonRetry.Q;

fbKoyo_PLCInputCoilsRx(sIPAddr:='i_sIPAddr', nTCPPort:=502, nQuantity:=32, nMBAddr:=8#6000, cbLength:=USINT_TO_UDINT(SIZEOF(anKoyo_PLC_CnBits)),  pDestAddr:=ADR(anKoyo_PLC_CnBits), tTimeout:=T#10S);

//run some error code for modbus
IF fbKoyo_PLCInputCoilsRx.bError THEN
    //if there's a modbus error, set all incoming bits to zero
    {analysis -41} //There are one-liners for resetting an array to zero but they don't comply with 61131
    FOR nIndex := 0 TO USINT_TO_INT(SIZEOF(anKoyo_PLC_CnBits))-1 DO //starts at 0
        anKoyo_PLC_CnBits[nIndex]:=0;
    END_FOR
    {analysis +41}
    bError := TRUE;

ELSIF ftReset.Q AND fbKoyo_PLCInputCoilsRx.cbRead > 0 THEN
    fbKoyo_PLCInputCoilsRx.bExecute := FALSE;
    bNoPLCResponse:= FALSE;
    bError := FALSE;

//more error code cause we didn't manage to read anything
ELSIF fbKoyo_PLCInputCoilsRx.cbRead = 0 THEN
    bError := TRUE;
    bNoPLCResponse:= TRUE;

END_IF

anPLCResponse := anKoyo_PLC_CnBits;

END_FUNCTION_BLOCK

// ---- POUs/Functions/TIME_TO_100NS.TcPOU
FUNCTION TIME_TO_100NS : ULINT
VAR_INPUT
    nTime : TIME;
END_VAR
VAR
END_VAR

TIME_TO_100NS := TIME_TO_ULINT(nTime)*10000;

END_FUNCTION

// ---- POUs/Hardware/FB_AnalogOutput.TcPOU
FUNCTION_BLOCK FB_AnalogOutput
(*
    Converts a real unit value (e.g., volts) to the integer needed for an analog output terminal.
    2019-10-09 Zachary Lentz
*)
VAR_INPUT
    // The real value to send to the output
    fReal: LREAL;
    // The maximum allowed real value for the connected hardware
    fSafeMax: LREAL;
    // The minimum allowed real value for the connected hardware
    fSafeMin: LREAL;
    // The number of bits correlated with the terminal's max output. This is not necessarily the resolution parameter.
    nTermBits: UINT;
    // The fReal value correlated with the terminal's max output
    fTermMax: LREAL;
    // The fReal value correlated with the terminal's min output
    fTermMin: LREAL;
END_VAR
VAR_OUTPUT
    // Connect this output to the terminal
    nRaw AT %Q*: INT;
END_VAR
VAR
    fScale: LREAL;
END_VAR

// Set the scaling from real to raw
IF fScale = 0 AND fTermMax > fTermMin THEN
    fScale := (EXPT(2, nTermBits) - 1) / (fTermMax - fTermMin);
END_IF

// Adjust real value to be within the limits
fReal := MIN(fReal, fSafeMax, fTermMax);
fReal := MAX(fReal, fSafeMin, fTermMin);

// Scale the output accordingly
nRaw := LREAL_TO_INT((fReal - fTermMin) * fScale);

END_FUNCTION_BLOCK

// ---- POUs/Hardware/FB_AnalogInput.TcPOU
FUNCTION_BLOCK FB_AnalogInput
(*
    Converts the integer from an analog input terminal to a real unit value (e.g., volts)
    2019-10-09 Zachary Lentz
*)
VAR_INPUT
    // Connect this input to the terminal
    iRaw AT %I*: DINT;
    // The number of bits correlated with the terminal's max value. This is not necessarily the resolution parameter.
    iTermBits: UINT;
    // The fReal value correlated with the terminal's max value
    fTermMax: LREAL;
    // The fReal value correlated with the terminal's min value
    fTermMin: LREAL;
    // Value to scale the end result to
    {attribute 'pytmc' := '
        pv: RES
        io: io
    '}
    fResolution : LREAL := 1;
    {attribute 'pytmc' := '
        pv: OFF
        io: io
    '}
    fOffset : LREAL;
END_VAR
VAR_OUTPUT
    // The real value read from the output
    {attribute 'pytmc' := '
        pv: VAL
        io: i
    '}
    fReal: LREAL;
END_VAR
VAR
    fScale: LREAL;
END_VAR

IF fScale = 0 AND fTermMax > fTermMin THEN
    fScale := (EXPT(2, iTermBits) - 1) / (fTermMax - fTermMin);
END_IF
IF fScale <> 0 THEN
    fReal := iRaw / fScale + fTermMin;
    fReal := fReal * fResolution + fOffset;
END_IF

END_FUNCTION_BLOCK

// ---- POUs/Hardware/FB_CoE_FastRead.TcPOU
FUNCTION_BLOCK FB_CoE_FastRead
(*
    Utility to repeatedly read a CoE parameter
    2019-10-09 Zachary Lentz

    In practice, it's impossible to read most CoE parameters every cycle,
    but this is a best effort and will work if the data is available
*)
VAR_INPUT
    // If TRUE we'll attempt a CoE read this cycle.
    bExecute: BOOL;
    // Link this to your terminal's drive reference variables under InfoData.
    stPlcDriveRef AT %I*: ST_PlcDriveRef;
    // Hexadecimal index of CoE, e.g. the 8010 in 8010:12
    nIndex: UINT;
    // Hexadecimal subindex of CoE, e.g. the 12 in 8010:12
    nSubIndex: BYTE;
    // Pointer to a value to fill with the result of the read, e.g. ADR(MyValue)
    pDstBuf: PVOID;
    // Data size of pDstBuf, e.g. SIZEOF(MyValue)
    cbBufLen: UINT;
END_VAR
VAR_OUTPUT
    // TRUE if the value was updated on this cycle.
    bNewValue: BOOL;
END_VAR
VAR
    fbRead: FB_CoERead_ByDriveRef;
    stDriveRef: ST_DriveRef;
    iLoop: INT;
    bInnerExec: BOOL;
END_VAR

stDriveRef.sNetId := F_CreateAmsNetId(stPlcDriveRef.aNetId);
stDriveRef.nSlaveAddr := stPlcDriveRef.nSlaveAddr;
stDriveRef.nDriveNo := stPlcDriveRef.nDriveNo;
stDriveRef.nDriveType := stPlcDriveRef.nDriveType;

bNewValue := FALSE;
IF bExecute THEN
    // You need to do this block 3 times per cycle to have a chance at always getting a read
    FOR iLoop:= 1 TO 3 DO
        fbRead(
            stDriveRef := stDriveRef,
            nIndex := nIndex,
            nSubIndex := nSubIndex,
            pDstBuf := pDstBuf,
            cbBufLen := cbBufLen,
            bExecute := bInnerExec,
            tTimeout := T#1s);

        IF bInnerExec AND NOT fbRead.bBusy AND NOT fbRead.bError THEN
            bInnerExec := FALSE;
            bNewValue := TRUE;
        ELSE
            bInnerExec := TRUE;
        END_IF
    END_FOR
END_IF

END_FUNCTION_BLOCK

// ---- POUs/Hardware/FB_ECATepics.TcPOU
FUNCTION_BLOCK FB_ECATepics
VAR_INPUT
    sNetId          : T_AmsNetId;
    nSlaveAddr      : UINT;
    sDeviceDesc		: T_MaxString := 'TERM #';
END_VAR
VAR_OUTPUT
END_VAR
VAR

    {attribute 'pytmc' := '
        pv: bCmdReqState
    '}

    bCmdReqState : BOOL;

    {attribute 'pytmc' := '
        pv: eReqState
    '}
    eReqState : E_ECAT_STATES;
    ePrevReqState : E_ECAT_STATES;

    {attribute 'pytmc' := '
        pv: eDevState
        io: o
        field: ZRSV MAJOR
        field: ONSV MAJOR
        field: TWSV MAJOR
        field: THSV MAJOR
        field: FRSV NO_ALARM
        field: FVSV MAJOR
    '}
    eDevState : E_ECAT_STATES;

    {attribute 'pytmc' := '
        pv: bError
        io: o
    '}
    bDevError : BOOL;

    {attribute 'pytmc' := '
        pv: sErrorMessage
        io: o
    '}
    sErrorMessage : STRING;

    {attribute 'pytmc' := '
        pv: sDESC
        io: io
    '}
    sDevDesc : STRING;

    fbsetSlaveState         : FB_EcSetSlaveState;
    fbgetSlaveState			: FB_EcGetSlaveState;
    fbgetStatusTimer : TON;
    bInit : BOOL := TRUE;

END_VAR

fbgetStatusTimer(PT:= T#500MS);

IF bInit THEN
    sDevDesc := sDeviceDesc;
    bInit := FALSE;
    fbgetStatusTimer.IN:= TRUE;
    ePrevReqState :=  eReqState;
END_IF

fbsetSlaveState(sNetId:=sNetId,
    nSlaveAddr:= nSlaveAddr,
    bExecute:= bCmdReqState,
    reqState:= eReqState);

fbgetSlaveState(sNetId:=sNetId,
    nSlaveAddr:= nSlaveAddr,
    bExecute:= fbgetStatusTimer.Q);

CASE fbgetSlaveState.state.deviceState OF
    EC_DEVICE_STATE_INIT:
        eDevState := E_ECAT_STATES.INIT;
    EC_DEVICE_STATE_PREOP:
        eDevState := E_ECAT_STATES.PREOP;
    EC_DEVICE_STATE_BOOTSTRAP:
        eDevState := E_ECAT_STATES.BOOTSTRAP;
    EC_DEVICE_STATE_SAFEOP:
        eDevState := E_ECAT_STATES.SAFEOP;
    EC_DEVICE_STATE_OP:
        eDevState := E_ECAT_STATES.OP;
    EC_DEVICE_STATE_ERROR:
        eDevState := E_ECAT_STATES.ERROR;
END_CASE

bDevError := fbsetSlaveState.bError;

IF bCmdReqState AND (bDevError OR (NOT fbsetSlaveState.bBusy)) THEN
    bCmdReqState := FALSE;
END_IF

CASE fbsetSlaveState.nErrId OF
    0: sErrorMessage := '';
    // --- Device errors (0x700 - 0x739) ---
    1792: sErrorMessage := 'ADSERR_DEVICE_ERROR - General device error.';
    1793: sErrorMessage := 'ADSERR_DEVICE_SRVNOTSUPP - Service is not supported by the server.';
    1794: sErrorMessage := 'ADSERR_DEVICE_INVALIDGRP - Invalid index group.';
    1795: sErrorMessage := 'ADSERR_DEVICE_INVALIDOFFSET - Invalid index offset.';
    1796: sErrorMessage := 'ADSERR_DEVICE_INVALIDACCESS - Reading or writing not permitted. ';
    1797: sErrorMessage := 'ADSERR_DEVICE_INVALIDSIZE - Parameter size not correct.';
    1798: sErrorMessage := 'ADSERR_DEVICE_INVALIDDATA - Invalid data values.';
    1799: sErrorMessage := 'ADSERR_DEVICE_NOTREADY - Device is not ready to operate.';
    1800: sErrorMessage := 'ADSERR_DEVICE_BUSY - Device is busy.';
    1801: sErrorMessage := 'ADSERR_DEVICE_INVALIDCONTEXT - Invalid operating system context.';
    1802: sErrorMessage := 'ADSERR_DEVICE_NOMEMORY - Insufficient memory.';
    1803: sErrorMessage := 'ADSERR_DEVICE_INVALIDPARM - Invalid parameter values.';
    1804: sErrorMessage := 'ADSERR_DEVICE_NOTFOUND - Not found (files, ...).';
    1805: sErrorMessage := 'ADSERR_DEVICE_SYNTAX - Syntax error in file or command.';
    1806: sErrorMessage := 'ADSERR_DEVICE_INCOMPATIBLE - Objects do not match.';
    1807: sErrorMessage := 'ADSERR_DEVICE_EXISTS - Object already exists.';
    1808: sErrorMessage := 'ADSERR_DEVICE_SYMBOLNOTFOUND - Symbol not found.';
    1809: sErrorMessage := 'ADSERR_DEVICE_SYMBOLVERSIONINVALID - Invalid symbol version. This can occur due to an online change. Create a new handle.';
    1810: sErrorMessage := 'ADSERR_DEVICE_INVALIDSTATE - Device (server) is in invalid state.';
    1811: sErrorMessage := 'ADSERR_DEVICE_TRANSMODENOTSUPP - AdsTransMode not supported.';
    1812: sErrorMessage := 'ADSERR_DEVICE_NOTIFYHNDINVALID - Notification handle is invalid.';
    1813: sErrorMessage := 'ADSERR_DEVICE_CLIENTUNKNOWN - Notification client not registered.';
    1814: sErrorMessage := 'ADSERR_DEVICE_NOMOREHDLS - No further handle available.';
    1815: sErrorMessage := 'ADSERR_DEVICE_INVALIDWATCHSIZE - Notification size too large.';
    1816: sErrorMessage := 'ADSERR_DEVICE_NOTINIT - Device not initialized.';
    1817: sErrorMessage := 'ADSERR_DEVICE_TIMEOUT - Device has a timeout.';
    1818: sErrorMessage := 'ADSERR_DEVICE_NOINTERFACE - Interface query failed.';
    1819: sErrorMessage := 'ADSERR_DEVICE_INVALIDINTERFACE - Wrong interface requested.';
    1820: sErrorMessage := 'ADSERR_DEVICE_INVALIDCLSID - Class ID is invalid.';
    1821: sErrorMessage := 'ADSERR_DEVICE_INVALIDOBJID - Object ID is invalid.';
    1822: sErrorMessage := 'ADSERR_DEVICE_PENDING - Request pending.';
    1823: sErrorMessage := 'ADSERR_DEVICE_ABORTED - Request is aborted.';
    1824: sErrorMessage := 'ADSERR_DEVICE_WARNING - Signal warning.';
    1825: sErrorMessage := 'ADSERR_DEVICE_INVALIDARRAYIDX - Invalid array index.';
    1826: sErrorMessage := 'ADSERR_DEVICE_SYMBOLNOTACTIVE - Symbol not active.';
    1827: sErrorMessage := 'ADSERR_DEVICE_ACCESSDENIED - Access denied.';
    1828: sErrorMessage := 'ADSERR_DEVICE_LICENSENOTFOUND - Missing license.';
    1829: sErrorMessage := 'ADSERR_DEVICE_LICENSEEXPIRED - License expired.';
    1830: sErrorMessage := 'ADSERR_DEVICE_LICENSEEXCEEDED - License exceeded.';
    1831: sErrorMessage := 'ADSERR_DEVICE_LICENSEINVALID - Invalid license.';
    1832: sErrorMessage := 'ADSERR_DEVICE_LICENSESYSTEMID - License problem: System ID is invalid.';
    1833: sErrorMessage := 'ADSERR_DEVICE_LICENSENOTIMELIMIT - License not limited in time.';
    1834: sErrorMessage := 'ADSERR_DEVICE_LICENSEFUTUREISSUE - Licensing problem: time in the future.';
    1835: sErrorMessage := 'ADSERR_DEVICE_LICENSETIMETOLONG - License period too long.';
    1836: sErrorMessage := 'ADSERR_DEVICE_EXCEPTION - Exception at system startup.';
    1837: sErrorMessage := 'ADSERR_DEVICE_LICENSEDUPLICATED - License file read twice.';
    1838: sErrorMessage := 'ADSERR_DEVICE_SIGNATUREINVALID - Invalid signature.';
    1839: sErrorMessage := 'ADSERR_DEVICE_CERTIFICATEINVALID - Invalid certificate.';
    1840: sErrorMessage := 'ADSERR_DEVICE_LICENSEOEMNOTFOUND - Public key not known from OEM.';
    1841: sErrorMessage := 'ADSERR_DEVICE_LICENSERESTRICTED - License not valid for this system ID.';
    1842: sErrorMessage := 'ADSERR_DEVICE_LICENSEDEMODENIED - Demo license prohibited.';
    1843: sErrorMessage := 'ADSERR_DEVICE_INVALIDFNCID - Invalid function ID.';
    1844: sErrorMessage := 'ADSERR_DEVICE_OUTOFRANGE - Outside the valid range.';
    1845: sErrorMessage := 'ADSERR_DEVICE_INVALIDALIGNMENT - Invalid alignment.';
    1846: sErrorMessage := 'ADSERR_DEVICE_LICENSEPLATFORM - Invalid platform level.';
    1847: sErrorMessage := 'ADSERR_DEVICE_FORWARD_PL - Context - forward to passive level.';
    1848: sErrorMessage := 'ADSERR_DEVICE_FORWARD_DL - Context - forward to dispatch level.';
    1849: sErrorMessage := 'ADSERR_DEVICE_FORWARD_RT - Context - forward to real-time.';

    ELSE
    sErrorMessage := 'Unknown ADS error code.';
END_CASE

IF fbgetStatusTimer.Q THEN
     fbgetStatusTimer.IN := FALSE; // reset timer
ELSE
    fbgetStatusTimer.IN := TRUE; // reset timer
END_IF

END_FUNCTION_BLOCK

// ---- POUs/Hardware/FB_EL6_Com.TcPOU
FUNCTION_BLOCK FB_EL6_Com
(*
    Communicate with a serial device connected to an EL6XXX
    2019-10-09 Zachary Lentz and Jackson Sheppard

    May contain assumptions about the device we wrote it for, potentially will need to be adjusted
*)
VAR_INPUT
    // Command to send to the serial device
    {attribute 'pytmc' := '
        pv: CMD
        io: io
    '}
    sCmd: STRING;

    // Pulse this to TRUE and back to FALSE when it's time to send
    {attribute 'pytmc' := '
        pv: SEND
        io: io
    '}
    bSend: BOOL;

    // Any static prefix to add before every sent message
    sSendPrefix: STRING;
    // Any static suffix to add after every sent message
    sSendSuffix: STRING;
    // Any static prefix to strip off of every recieved message
    sRecvPrefix: STRING;
    // Any static suffic to strip off of every recieved message
    sRecvSuffix: STRING;
    tTimeout: TIME := T#1S;
END_VAR
VAR_IN_OUT
    stIn_EL6: EL6inData22B;
    stOut_EL6: EL6outData22B;
END_VAR
VAR_OUTPUT
    // The response recieved from the serial device
    {attribute 'pytmc' := '
        pv: RESP
        io: input
    '}
    sResponse: STRING;

    // This is set to TRUE after recieving a response
    {attribute 'pytmc' := '
        pv: DONE
        io: input
    '}
    bDone: BOOL;

    {attribute 'pytmc' := '
        pv: ERR:SER
        io: input
    '}
    eSerialLineErrorID: ComError_t;

    {attribute 'pytmc' := '
        pv: ERR:SEND
        io: input
    '}
    eSendErrorID: ComError_t;

    {attribute 'pytmc' := '
        pv: ERR:RECV
        io: input
    '}
    eRecvErrorID: ComError_t;
END_VAR
VAR
    // Communication Buffers
    stTxBuffer: ComBuffer;
    stRxBuffer: ComBuffer;
    fbClearComBuffer: ClearComBuffer;

    // Parameters for PLC -> EL6
    fbEL6Ctrl: SerialLineControl;
    bEL6CtrlError: BOOL;
    eEL6CtrlErrorID: ComError_t;

    // Parameters for EL6 -> Serial Device
    fbSend: SendString;
    bSendBusy: BOOL;
    eLastSendErrorID: ComError_t;
    fbReceive: ReceiveString;
    sReceivedString: STRING;
    sLastReceivedString: STRING;
    bStringReceived: BOOL;
    bReceiveBusy: BOOL;
    bReceiveError: BOOL;
    eReceiveErrorID: ComError_t;
    bReceiveTimeout: BOOL;
    nReceiveCounter: UDINT;
    nSendCounter: UDINT;
    sStringToSend: STRING;
    fbFormatString: FB_FormatString;

    // Parameters for state-machine implementation
    nStep: INT := 0;
END_VAR

fbEL6Ctrl(
    Mode:= SERIALLINEMODE_EL6_22B,
    pComIn:= ADR(stIn_EL6),
    pComOut:= ADR(stOut_EL6),
    SizeComIn:= UINT_TO_INT(SIZEOF(stIn_EL6)),
    Error=> ,
    ErrorID=> eSerialLineErrorID,
    TxBuffer:= stTxBuffer,
    RxBuffer:= stRxBuffer );
IF fbEL6Ctrl.Error THEN
    bEL6CtrlError := TRUE;
    eEL6CtrlErrorID := fbEL6Ctrl.ErrorID;
END_IF
IF bSend THEN
    nStep := 10;
    bSend := FALSE;
    bDone := FALSE;
END_IF
// Attempt at solution that sends one command at a time, not on constant loop
CASE nStep OF
    0:
        ; // idle
    10:
        // Clear buffers in case any lingering data
        fbClearComBuffer(Buffer:=stTxBuffer);
        fbClearComBuffer(Buffer:=stRxBuffer);
        // Prepare string to send
        sStringToSend := CONCAT(sSendPrefix, CONCAT(sCmd, sSendSuffix));
        // Send string
        fbSend(	SendString:= sStringToSend,
                TXbuffer:= stTxBuffer,
                Busy=> bSendBusy,
                Error=> eSendErrorID);
        IF fbSend.Error <> COMERROR_NOERROR THEN
            eLastSendErrorID := fbSend.Error;
        ELSE
            nSendCounter := nSendCounter + 1;
        END_IF
        nStep := nStep + 10;
    20:
        // Finish sending String
        IF fbSend.Busy THEN
            fbSend(	SendString:= sStringToSend,
                    TXbuffer:= stTxBuffer,
                    Busy=> bSendBusy,
                    Error=> eSendErrorID);
            IF fbSend.Error <> COMERROR_NOERROR THEN
                eLastSendErrorID := fbSend.Error;
            ELSE
                nSendCounter := nSendCounter + 1;
            END_IF
        ELSE
            nStep := nStep + 10;
        END_IF
    30:
        // Get Reply
        fbReceive(
            Prefix:= sRecvPrefix,
            Suffix:= sRecvSuffix,
            Timeout:= tTimeout,
            ReceivedString:= sReceivedString,
            RXbuffer:= stRxBuffer,
            StringReceived=> bStringReceived,
            Busy=> bReceiveBusy,
            Error=> eRecvErrorID,
            RxTimeout=> bReceiveTimeout );
        IF fbReceive.Error <> COMERROR_NOERROR THEN
            eReceiveErrorID := fbReceive.Error;
        END_IF
        IF bStringReceived THEN
            nReceiveCounter := nReceiveCounter + 1;
            // Check for response
            IF FIND(sReceivedString, sStringToSend)=0 THEN
                sResponse := sReceivedString;
                bDone := TRUE;
                nStep := 0;
            END_IF
        END_IF
END_CASE

END_FUNCTION_BLOCK

// ---- POUs/Hardware/FB_LED.TcPOU
FUNCTION_BLOCK FB_LED
(*
    Reads a percentage of illumination determined by the user and converts it to a raw value
    to send to the terminal output via the FB_AnalogOutput.

    The determination of the full scale raw value (FSV) is calculated via the iTermBits,
    which is setup as an input variable to be set according to the situation. This value
    is bounded by the FSV of the terminal set by the Beckhoff architecture: (2^15 - 1) = 32767.

    Through the configurable max raw value sent to the terminal output, this LED function block
    is applicable to a wider variety of hardware: whether it be simple Analog Voltage control,
    PWM voltage output, or current controlled output.

    As an initial application, this FB will be instituted for systems of vaccum chamber LED
    illuminators on TMO endstations, which are rated for 12 V max. They will be dimmed via the
    EL2502 terminal 24 V PWM output voltage control from 0-50% duty cycle.

    2022-5-03 Maarten Thomas-Bosum
*)
VAR_INPUT
    {attribute 'pytmc' := '
        pv: NAME
        io: io
        field: DESC Descriptive name for the LED
        autosave_pass0: VAL DESC
    '}
    sLedName : STRING;

    nTermBits : UINT;

    {attribute 'pytmc' := '
        pv: ILL:PCT
        field: EGU %
    '}
    fIlluminatorPercent: LREAL;

    {attribute 'pytmc' := '
        pv: PWR
        field: ZNAM OFF
        field: ONAM ON
    '}
    bLedPower AT %Q*: BOOL;
END_VAR
VAR
    nIlluminatorINT AT %Q*: INT;
    fbSetIllPercent: FB_AnalogOutput;
END_VAR

// Illuminator conversion to percentage
fbSetIllPercent(
    fReal:=fIlluminatorPercent,
    fSafeMax:=100,
    fSafeMin:=0,
    nTermBits:=nTermBits,
    fTermMax:=100,
    fTermMin:=0,
    nRaw=>nIlluminatorINT);

IF  fIlluminatorPercent > 0 THEN
    bLedPower := TRUE;
ELSE
    bLEDPower := FALSE;
END_IF

END_FUNCTION_BLOCK

// ---- POUs/Hardware/FB_ThermoCouple.TcPOU
FUNCTION_BLOCK FB_ThermoCouple
(*
    Deprecated as of 2020-03-02, please use FB_TempSensor instead
    2019-10-09 Zachary Lentz
*)
{warning 'Function Block FB_ThermoCouple is deprecated and may be removed in a future release'}
VAR_INPUT
    // Ratio between raw value and actual temperature. Default is 10 for 10 steps per degree (or 0.1 degree resolution)
    nScale: INT := 10;
END_VAR
VAR_OUTPUT
    {attribute 'pytmc' := '
        pv: STC:TEMP
        io: input
    '}
    fTemp: LREAL;

    {attribute 'pytmc' := '
        pv: STC:CONN
        io: input
        field: ONAM Connected
        field: ZNAM Disconnected
    '}
    bConnected: BOOL;

    {attribute 'pytmc' := '
        pv: STC:ERR
        io: input
    '}
    bError AT %I*: BOOL;

    bUnderrange AT %I*: BOOL;
    bOverrange AT %I*: BOOL;
END_VAR
VAR
    nRaw AT %I*: INT;
END_VAR

// The manual states that we are disconnected if we are both overrange and in an error state
bConnected := NOT (bOverrange AND bError);
fTemp := INT_TO_LREAL(nRaw) / nScale;

END_FUNCTION_BLOCK

// ---- POUs/Hardware/FB_TempSensor.TcPOU
FUNCTION_BLOCK FB_TempSensor
(*
    Handles scaling and default diagnostics for temperature sensors,
    such as thermocouples, RTDs, and others.
    2020-03-02 Zachary Lentz
*)
VAR_INPUT
    // Resolution parameter from the Beckhoff docs. Default is 0.1 for 0.1 degree resolution
    fResolution: LREAL := 0.1;
END_VAR
VAR_OUTPUT
    {attribute 'pytmc' := '
        pv: TEMP
        io: input
        field: EGU C
        field: PREC 2
    '}
    fTemp: LREAL;

    {attribute 'pytmc' := '
        pv: CONN
        io: input
        field: ONAM Connected
        field: ZNAM Disconnected
    '}
    bConnected: BOOL;

    {attribute 'pytmc' := '
        pv: ERR
        io: input
        field: ONAM True
        field: ZNAM False
    '}
    bError AT %I*: BOOL := TRUE;

    bUnderrange AT %I*: BOOL;
    bOverrange AT %I*: BOOL;
END_VAR
VAR
    nRaw AT %I*: INT;
END_VAR

// The manual states that we are disconnected if we are both overrange and in an error state
bConnected := NOT (bOverrange AND bError);
fTemp := INT_TO_LREAL(nRaw) * fResolution;

END_FUNCTION_BLOCK

// ---- POUs/Logger/SYSTEM_TIME_TO_RFC3339.TcPOU
//Converts Beckhoff PLC SYSTEMTIME to RFC3339 time format as a string
{attribute 'naming' := 'omit'}
{attribute 'analysis' := '-23'}
FUNCTION SYSTEM_TIME_TO_RFC3339 : STRING(255)
VAR_INPUT
    {attribute 'naming' := 'omit'}
    tCurrentTime	:	TIMESTRUCT; //TIMESTRUCT Time to convert to RFC3339
END_VAR
VAR
END_VAR

SYSTEM_TIME_TO_RFC3339 := CONCAT(REPLACE(SYSTEMTIME_TO_STRING(tCurrentTime), 'T', 1, 11), 'Z');

END_FUNCTION
